// TIA Portal V16 export
// export: Created 2024-09-05T17:40:13.4646114Z, ExportSetting WithDefaults, DisplayName Totally Integrated Automation Portal, DisplayVersion V16 Update 6, DisplayName TIA Portal Version Control Interface, DisplayVersion V16 Update 2, DisplayName TIA Portal Openness, DisplayVersion V16 Update 6, DisplayName STEP 7 Professional, DisplayVersion V16 Update 6, DisplayName STEP 7 Safety, DisplayVersion V16, DisplayName WinCC Advanced, DisplayVersion V16 Update 6
TYPE "UDT_PositionData"
// stored: IsFailsafeCompliant false
   STRUCT
      PartPresent : Bool;
      PartNOK : Bool;
      PartErrors : Array[0..255] of Bool;
      Reference : Int;
      FinishedOperations : Array[0..15] of Bool;
      StFinished : Array[0..15] of Bool;
      Scan : String[30];
      IJCType : Int;   // 0 - no ijc; 1 - Standart IJC; 2 - P variant; 3 - downgrade mode
      CodeReadings : Struct   // Label code readings
         SideMemberLH : String[128];
         SideMemberRH : String[128];
         RearTube : String[128];
         FrontTube : String[128];
      END_STRUCT;
   END_STRUCT;
END_TYPE
